// TIA Portal V20 export
// export: Created 2025-12-01T14:56:10.1501103Z, ExportSetting None, DisplayName Totally Integrated Automation Portal, DisplayVersion V20 Update 3, DisplayName TIA Portal Openness, DisplayVersion V20 Update 3, DisplayName TIA Portal Version Control Interface, DisplayVersion V20 Update 3, DisplayName STEP 7 Professional, DisplayVersion V20 Update 3, DisplayName STEP 7 Safety, DisplayVersion V20 Update 2, DisplayName WinCC Basic/Comfort/Advanced, DisplayVersion V20 Update 3, DisplayName WinCC Professional, DisplayVersion V20 Update 3, DisplayName WinCC Unified, DisplayVersion V20 Update 3
TYPE "LPNDR_typePortInformation"
   STRUCT
      numbersOfPeers : Byte;
      lineDelay : UDInt;
      peerMacAdress : Array[0..5] of Byte;
      peerNameofStation : String;
      peerPortName : String[14];
      dataRate : String[5];   // Bit/sec
      mediaType : USInt;   // 0=unknown, 1=Cooper cable, 2 = Fiber optic cable, 3=Radio communication
      portDiagnostic { S7_SetPoint := 'True'} : "LPNDR_typePortLinkState";
   END_STRUCT;
END_TYPE
